% RSLogix 500 project PLC_1_LAB6-1-TEST.RSS, saved by version 12.00.00.00 %
PROJECT "UNTITLED"    % processor: Bul.1763 MicroLogix 1100 Series B %

PROGRAM FILES
  LAD 2   2 rungs

DATA FILES
  O0 OUTPUT  5 elements
  I1 INPUT  6 elements
  S2 STATUS  66 elements
  B3 BINARY  1 elements
  T4 TIMER  2 elements
  C5 COUNTER  1 elements
  R6 CONTROL  1 elements
  N7 INTEGER  1 elements
  F8 FLOAT  1 elements

LADDER 2
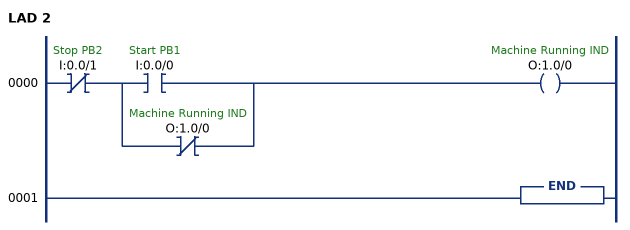
% Rung: 0 %
SOR XIO I:0.0/1 BST XIC I:0.0/0 NXB XIO O:1.0/0 BND OTE O:1.0/0 EOR
%   I:0.0/1  PB2  "Stop" %
%   I:0.0/0  PB1  "Start" %
%   O:1.0/0  IND  "Machine Running" %
% Rung: 1 %
SOR END EOR

OTHER DOCUMENTED ADDRESSES
  C5:0  CBT  "Bottle Counter"
  T4:0  "Filled Soda"
  T4:1  "Foam To subside"
  XIC  
  XIO  

DATA TABLE (non-zero values as saved)
DATA T4
% .PRE .ACC %
% T4:0 % 740 0
DATA C5
% .PRE .ACC %
% C5:0 % 3 0
